FUNCTION_BLOCK Recipe_11020_TequilaSunrise
VAR_INPUT
	TaskID	: 	LREAL;
	Execute :	BOOL;
	Parameter	: ARRAY [1..UserParameterCnt] OF DUT_RECIPE_USERPARAMETERINPUT;
END_VAR
VAR_OUTPUT
	RecipeDone	: BOOL;
	RecipeInfo	: DUT_RECIPEOFFER;
	InitDone	: BOOL;
END_VAR
VAR	
	Done		: BOOL;
	Priority	: INT;
	
END_VAR

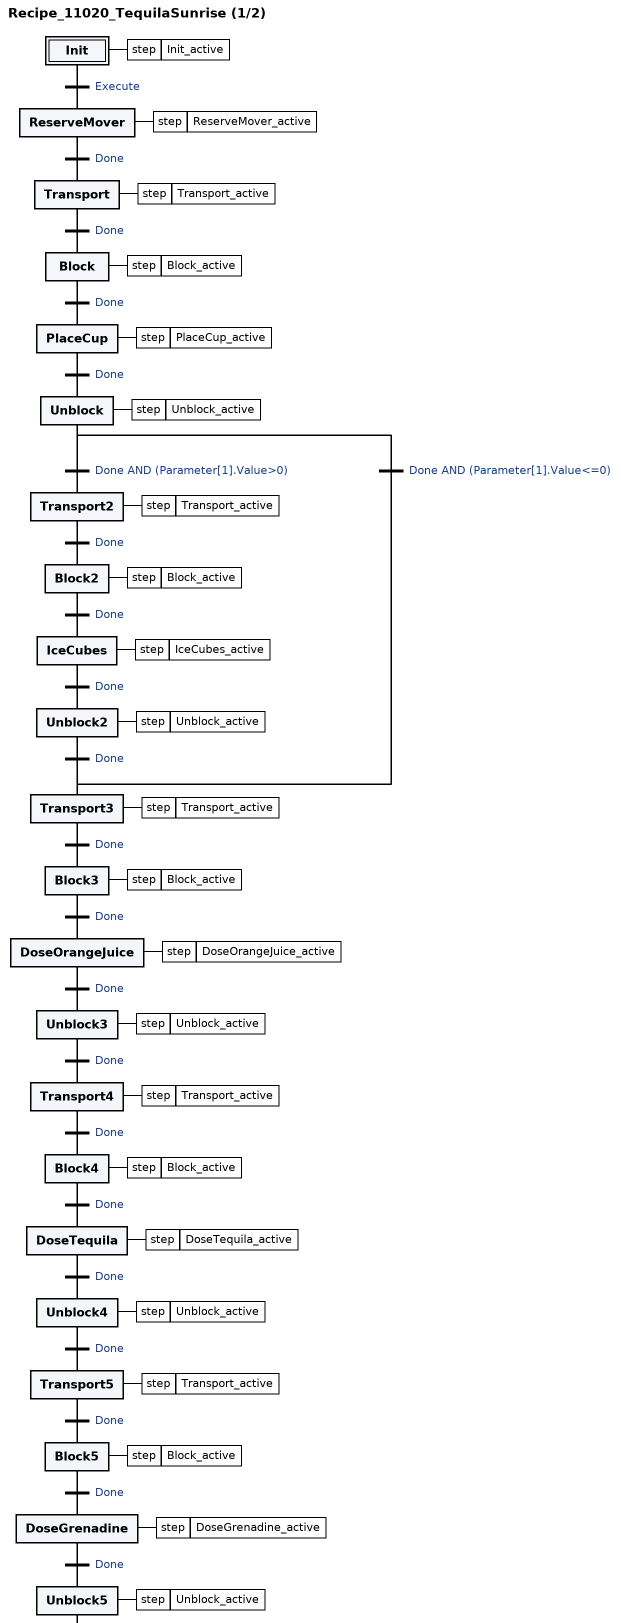
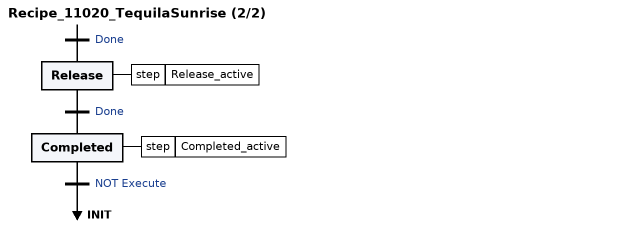
INITIAL_STEP Init:
    Init_active(N);  // step action
END_STEP
TRANSITION FROM Init TO ReserveMover
    := Execute;
END_TRANSITION
STEP ReserveMover:
    ReserveMover_active(N);  // step action
END_STEP
TRANSITION FROM ReserveMover TO Transport
    := Done;
END_TRANSITION
STEP Transport:
    Transport_active(N);  // step action
END_STEP
TRANSITION FROM Transport TO Block
    := Done;
END_TRANSITION
STEP Block:
    Block_active(N);  // step action
END_STEP
TRANSITION FROM Block TO PlaceCup
    := Done;
END_TRANSITION
STEP PlaceCup:
    PlaceCup_active(N);  // step action
END_STEP
TRANSITION FROM PlaceCup TO Unblock
    := Done;
END_TRANSITION
STEP Unblock:
    Unblock_active(N);  // step action
END_STEP
TRANSITION FROM Unblock TO Transport2
    := Done AND (Parameter[1].Value>0);
END_TRANSITION
STEP Transport2:
    Transport_active(N);  // step action
END_STEP
TRANSITION FROM Transport2 TO Block2
    := Done;
END_TRANSITION
STEP Block2:
    Block_active(N);  // step action
END_STEP
TRANSITION FROM Block2 TO IceCubes
    := Done;
END_TRANSITION
STEP IceCubes:
    IceCubes_active(N);  // step action
END_STEP
TRANSITION FROM IceCubes TO Unblock2
    := Done;
END_TRANSITION
STEP Unblock2:
    Unblock_active(N);  // step action
END_STEP
TRANSITION FROM Unblock2 TO Transport3
    := Done;
END_TRANSITION
TRANSITION FROM Unblock TO Transport3
    := Done AND (Parameter[1].Value<=0);
END_TRANSITION
STEP Transport3:
    Transport_active(N);  // step action
END_STEP
TRANSITION FROM Transport3 TO Block3
    := Done;
END_TRANSITION
STEP Block3:
    Block_active(N);  // step action
END_STEP
TRANSITION FROM Block3 TO DoseOrangeJuice
    := Done;
END_TRANSITION
STEP DoseOrangeJuice:
    DoseOrangeJuice_active(N);  // step action
END_STEP
TRANSITION FROM DoseOrangeJuice TO Unblock3
    := Done;
END_TRANSITION
STEP Unblock3:
    Unblock_active(N);  // step action
END_STEP
TRANSITION FROM Unblock3 TO Transport4
    := Done;
END_TRANSITION
STEP Transport4:
    Transport_active(N);  // step action
END_STEP
TRANSITION FROM Transport4 TO Block4
    := Done;
END_TRANSITION
STEP Block4:
    Block_active(N);  // step action
END_STEP
TRANSITION FROM Block4 TO DoseTequila
    := Done;
END_TRANSITION
STEP DoseTequila:
    DoseTequila_active(N);  // step action
END_STEP
TRANSITION FROM DoseTequila TO Unblock4
    := Done;
END_TRANSITION
STEP Unblock4:
    Unblock_active(N);  // step action
END_STEP
TRANSITION FROM Unblock4 TO Transport5
    := Done;
END_TRANSITION
STEP Transport5:
    Transport_active(N);  // step action
END_STEP
TRANSITION FROM Transport5 TO Block5
    := Done;
END_TRANSITION
STEP Block5:
    Block_active(N);  // step action
END_STEP
TRANSITION FROM Block5 TO DoseGrenadine
    := Done;
END_TRANSITION
STEP DoseGrenadine:
    DoseGrenadine_active(N);  // step action
END_STEP
TRANSITION FROM DoseGrenadine TO Unblock5
    := Done;
END_TRANSITION
STEP Unblock5:
    Unblock_active(N);  // step action
END_STEP
TRANSITION FROM Unblock5 TO Release
    := Done;
END_TRANSITION
STEP Release:
    Release_active(N);  // step action
END_STEP
TRANSITION FROM Release TO Completed
    := Done;
END_TRANSITION
STEP Completed:
    Completed_active(N);  // step action
END_STEP
TRANSITION FROM Completed TO INIT
    := NOT Execute;
END_TRANSITION

ACTION IceCubes_active:
Done := FALSE;

ExecuteSkill.SkillID 			:= 1401;
ExecuteSkill.SkillName	 		:= 'Dispense Ice Cubes';
ExecuteSkill.Parameter[1].ID 	:= 1;
ExecuteSkill.Parameter[1].Name 	:= 'Amount';
ExecuteSkill.Parameter[1].Value := Parameter[1].Value;
ExecuteSkill();
Done := TRUE;
END_ACTION

ACTION Completed_active:
RecipeDone := TRUE;
Done := FALSE;
END_ACTION

ACTION Init_active:
RecipeDone := FALSE;

// Initialisation of Recipe Parameters an name etc
RecipeInfo.Name := 'Tequila Sunrise';
RecipeInfo.Description := 'This Recipe produces a simple yolo #sunrise';
RecipeInfo.Dummy := FALSE;
RecipeInfo.RecipeID := 10020;
Initdone := TRUE;

//Parameter 1:
(*
	RecipeInfo.UserParameter[1].Dummy 		:= 
	RecipeInfo.UserParameter[1].Default		:=
	RecipeInfo.UserParameter[1].Description	:=
	RecipeInfo.UserParameter[1].MaxValue	:=
	RecipeInfo.UserParameter[1].MinValue	:=
	RecipeInfo.UserParameter[1].Name		:=
	RecipeInfo.UserParameter[1].Unit		:=
*)
//Parameter 2:

(*
	RecipeInfo.UserParameter[2].Dummy 		:= 
	RecipeInfo.UserParameter[2].Default		:=
	RecipeInfo.UserParameter[2].Description	:=
	RecipeInfo.UserParameter[2].MaxValue	:=
	RecipeInfo.UserParameter[2].MinValue	:=
	RecipeInfo.UserParameter[2].Name		:=
	RecipeInfo.UserParameter[2].Unit		:=
*)

//Parameter 3:

(*
	RecipeInfo.UserParameter[3].Dummy 		:= 
	RecipeInfo.UserParameter[3].Default		:=
	RecipeInfo.UserParameter[3].Description	:=
	RecipeInfo.UserParameter[3].MaxValue	:=
	RecipeInfo.UserParameter[3].MinValue	:=
	RecipeInfo.UserParameter[3].Name		:=
	RecipeInfo.UserParameter[3].Unit		:=
*)

//Parameter 4:

(*
	RecipeInfo.UserParameter[4].Dummy 		:= 
	RecipeInfo.UserParameter[4].Default		:=
	RecipeInfo.UserParameter[4].Description	:=
	RecipeInfo.UserParameter[4].MaxValue	:=
	RecipeInfo.UserParameter[4].MinValue	:=
	RecipeInfo.UserParameter[4].Name		:=
	RecipeInfo.UserParameter[4].Unit		:=
*)


//Parameter 5:

(*
	RecipeInfo.UserParameter[5].Dummy 		:= 
	RecipeInfo.UserParameter[5].Default		:=
	RecipeInfo.UserParameter[5].Description	:=
	RecipeInfo.UserParameter[5].MaxValue	:=
	RecipeInfo.UserParameter[5].MinValue	:=
	RecipeInfo.UserParameter[5].Name		:=
	RecipeInfo.UserParameter[5].Unit		:=
*)
END_ACTION

ACTION ReserveMover_active:
Done := FALSE;


ExecuteSkill.SkillID := 1310;
ExecuteSkill.SkillName	 := 'Reserve Mover';
ExecuteSkill.Parameter[1].ID := 1;
ExecuteSkill.Parameter[1].Name := 'TaskID';
ExecuteSkill.Parameter[1].Value := TaskID;
ExecuteSkill();

Done := TRUE;
END_ACTION

ACTION DoseGrenadine_active:
Done := FALSE;

ExecuteSkill.SkillID 			:= 1012;
ExecuteSkill.SkillName	 		:= 'Dose Orange Juice';
ExecuteSkill.Parameter[1].ID 	:= 1;
ExecuteSkill.Parameter[1].Name 	:= 'Amount';
ExecuteSkill.Parameter[1].Value := 12;//[ml]

ExecuteSkill.Parameter[2].ID 	:= 2;
ExecuteSkill.Parameter[2].Name 	:= 'SpeedFaktor';
ExecuteSkill.Parameter[2].Value := 0.5;//[ml]


ExecuteSkill();
Done := TRUE;
END_ACTION

ACTION Release_active:
Done := FALSE;


ExecuteSkill.SkillID 			:= 1311;
ExecuteSkill.SkillName	 		:= 'Release Mover';
ExecuteSkill.Parameter[1].ID 	:= 1;
ExecuteSkill.Parameter[1].Name 	:= 'TaskID';
ExecuteSkill.Parameter[1].Value := TaskID;
ExecuteSkill();

Done := TRUE;
END_ACTION

ACTION DoseOrangeJuice_active:
Done := FALSE;

ExecuteSkill.SkillID 			:= 1011;
ExecuteSkill.SkillName	 		:= 'Dose Orange Juice';
ExecuteSkill.Parameter[1].ID 	:= 1;
ExecuteSkill.Parameter[1].Name 	:= 'Amount';
ExecuteSkill.Parameter[1].Value := 133;//[ml]
ExecuteSkill();
Done := TRUE;
END_ACTION

ACTION Transport_active:
Done := FALSE;

//Skill auswählen
ExecuteSkill.SkillID 		:= 1320;
ExecuteSkill.SkillName	 	:= 'Transport Mover';

//Geschwindigkeit setzen
ExecuteSkill.Parameter[1].ID := 3;
ExecuteSkill.Parameter[1].Name := 'Velocity';
ExecuteSkill.Parameter[1].Value := 3000;


ExecuteSkill();

Done := ExecuteSkill.Done;
END_ACTION

ACTION Block_active:
Done := FALSE;

//Skill auswählen
ExecuteSkill.SkillID := 1315;
ExecuteSkill.SkillName	 := 'Block Mover';

//Parameter setzen
ExecuteSkill.Parameter[1].ID := 1;
ExecuteSkill.Parameter[1].Name := 'TaskID';
ExecuteSkill.Parameter[1].Value := TaskID;

//Skill hinzufügen
ExecuteSkill();


Done := TRUE;
END_ACTION

ACTION Unblock_active:
Done := FALSE;

//Skill auswählen
ExecuteSkill.SkillID := 1316;
ExecuteSkill.SkillName	 := 'Unblock Mover';

//Parameter setzen
ExecuteSkill.Parameter[1].ID := 1;
ExecuteSkill.Parameter[1].Name := 'TaskID';
ExecuteSkill.Parameter[1].Value := TaskID;

//Skill hinzufügen
ExecuteSkill();


Done := TRUE;
END_ACTION

ACTION PlaceCup_active:
Done := FALSE;

ExecuteSkill.SkillID 			:= 1402;
ExecuteSkill.SkillName	 		:= 'Place Cup';

ExecuteSkill();
Done := TRUE;
END_ACTION

ACTION DoseTequila_active:
Done := FALSE;

ExecuteSkill.SkillID 			:= 1009;
ExecuteSkill.SkillName	 		:= 'Dose Tequila';
ExecuteSkill.Parameter[1].ID 	:= 1;
ExecuteSkill.Parameter[1].Name 	:= 'Amount';
ExecuteSkill.Parameter[1].Value := 50;//[ml]
ExecuteSkill();
Done := TRUE;
END_ACTION

END_FUNCTION_BLOCK

(* stored: Version 1.1.0.1, ProductVersion 3.1.0.25
   POU Recipe_11020_TequilaSunrise: Id {4e40c0a0-115b-4076-927e-6934e19ac623}
   Action IceCubes_active: Id {2bb08cb9-10e3-4955-aa38-578d60e86f9f}
   Action Completed_active: Id {2d242d2c-c97c-4d3b-a4f6-ec15aae6927f}
   Action Init_active: Id {329cde14-f730-45c4-835b-52dec4f51216}
   Action ReserveMover_active: Id {41657dc0-1719-413d-89a9-859567b923fb}
   Action DoseGrenadine_active: Id {484241c1-4b2d-4c76-9317-cf69db590ee4}
   Action Release_active: Id {679e20af-6e7c-461d-b5fc-63e10b8a78d0}
   Action DoseOrangeJuice_active: Id {a89c5ea6-8498-4380-be50-b6104ecbbaa4}
   Action Transport_active: Id {aad03207-30e7-47cb-a862-f5217cfed0b6}
   Action Block_active: Id {b15ef0f3-29f0-4c02-a0ba-6b7f76a0ff4f}
   Action Unblock_active: Id {dd7fd46f-74cb-418c-9a17-60496188e528}
   Action PlaceCup_active: Id {df25d159-458f-4cbf-bf2a-a7f3a635e14d}
   Action DoseTequila_active: Id {e117e2a5-94ed-4022-bf60-25c865970b61} *)
